// TIA Portal V19 export
TYPE "Positioning_DOL_Machine_Wng"
// stored: Access Published
   STRUCT
      NotAutReady : Bool;   // Machine is NOT ready for automatic start
      MissingCnd_Minus : Bool;   // Lack of conditions for movement in negative direction
      MissingCnd_Plus : Bool;   // Lack of conditions for movement in positive direction
      Ax_NotHomed { ExternalAccessible := 'False'; ExternalVisible := 'False'; ExternalWritable := 'False'} : Bool;   // Axis is not homed / referenced
      Ax : "OOAx_Wng";   // ON-OFF AXIS
      S120 : Struct   // SINAMICS S120
         Drive : Bool;   // Warning presence
      END_STRUCT;
   END_STRUCT;
   // // Ax.SwLimitMinus : Negative software limit reached / exceeded.
   // // Ax.SwLimitPlus : Positive software limit reached / exceeded.
END_TYPE
